// TIA Portal V18 export
DATA_BLOCK "IO_MAP"   // DB1
{ S7_Optimized_Access := 'FALSE' }
VERSION : 0.1
// stored: AutoNumber true, DBAccessibleFromOPCUA true, IsOnlyStoredInLoadMemory false, IsWriteProtectedInAS false
   VAR
      D_IN { S7_SetPoint := 'True'} : "DI";
      D_OUT { S7_SetPoint := 'True'} : "DO";
      A_OUT { S7_SetPoint := 'True'} : "AO";
      A_IN { S7_SetPoint := 'True'} : "AI";
      RTD { S7_SetPoint := 'True'} : "RTD";
   END_VAR
BEGIN
END_DATA_BLOCK
